Staubli VAL3: recordPowerDown.pgx

public program recordPowerDown()
begin
  // record the powerDown point
  pTollerance=here(flange,world)
end
